TYPE aT_Pump :
STRUCT
	SetSpeed: LREAL;
	Pressure: LREAL;
	Flow: LREAL;
END_STRUCT
END_TYPE

(* stored: Version 1.1.0.1, ProductVersion 3.1.4024.4
   DUT aT_Pump: Id {5ca94a6f-7963-44d6-b323-373c57e7b6f2} *)
